{attribute 'qualified_only'}
VAR_GLOBAL
    fbScatteringFactors : FB_ScatteringFactorLUT;
END_VAR

(* stored: Version 1.1.0.1, ProductVersion 3.1.4022.18
   GVL GVL_Physics: Id {7147a988-93cf-4830-ac6b-3807273ff8ec} *)
